FUNCTION_BLOCK ASR_CLIENT_0 (* Trigger 2 independent remote OPC-UA method calls via CLIENT_0, driven by an ASR adapter Socket (Set/Reset) *)
  (* Standard: 61499-2; Description: Copyright (c) 2026 HR Agrartechnik GmbH This program and the accompanying materials are made available under the terms of the Eclipse Public License 2.0 which is available at https://www.eclipse.org/legal/epl-2.0/ SPDX-License-Identifier: EPL-2.0 *)
  (* Version 1.0, 2026-09-03, Franz Höpfinger, HR Agrartechnik GmbH, initial API and implementation and/or initial documentation *)
  PACKAGE adapter::net;
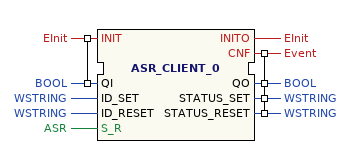
  EVENT_INPUT
    INIT : EInit WITH QI; (* Initialization *)
  END_EVENT
  EVENT_OUTPUT
    INITO : EInit; (* Initialization Confirm *)
    CNF WITH QO, STATUS_SET, STATUS_RESET; (* QO/STATUS updated *)
  END_EVENT
  VAR_INPUT
    QI : BOOL;
    ID_SET : WSTRING; (* Remote-Methodenadresse fuer den Set-Aufruf *)
    ID_RESET : WSTRING; (* Remote-Methodenadresse fuer den Reset-Aufruf *)
  END_VAR
  VAR_OUTPUT
    QO : BOOL; (* TRUE nur wenn SET_CLIENT und RESET_CLIENT aktuell beide QO=TRUE melden *)
    STATUS_SET : WSTRING; (* STATUS von SET_CLIENT *)
    STATUS_RESET : WSTRING; (* STATUS von RESET_CLIENT *)
  END_VAR
  SOCKETS
    S_R : adapter::types::unidirectional::ASR; (* Set/Reset *)
  END_SOCKETS
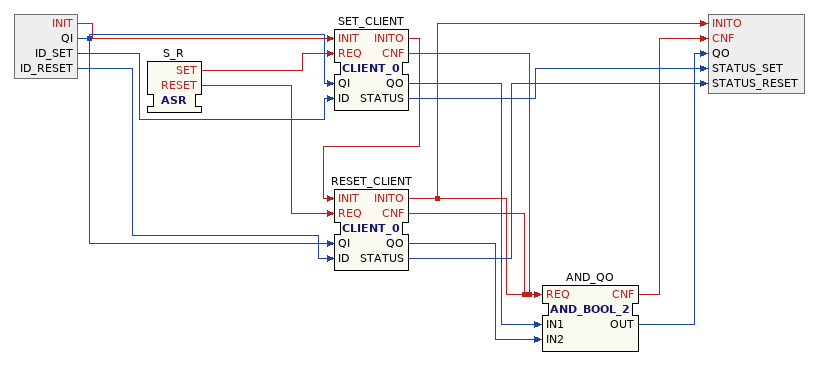
  FBS
    SET_CLIENT : iec61499::net::CLIENT_0;
    RESET_CLIENT : iec61499::net::CLIENT_0;
    AND_QO : iec61131::booleanOperators::AND_BOOL_2;
  END_FBS
  EVENT_CONNECTIONS
    INIT TO SET_CLIENT.INIT;
    SET_CLIENT.INITO TO RESET_CLIENT.INIT;
    RESET_CLIENT.INITO TO INITO;
    RESET_CLIENT.INITO TO AND_QO.REQ;
    S_R.SET TO SET_CLIENT.REQ;
    S_R.RESET TO RESET_CLIENT.REQ;
    SET_CLIENT.CNF TO AND_QO.REQ;
    RESET_CLIENT.CNF TO AND_QO.REQ;
    AND_QO.CNF TO CNF;
  END_CONNECTIONS
  DATA_CONNECTIONS
    QI TO SET_CLIENT.QI;
    QI TO RESET_CLIENT.QI;
    ID_SET TO SET_CLIENT.ID;
    ID_RESET TO RESET_CLIENT.ID;
    SET_CLIENT.QO TO AND_QO.IN1;
    RESET_CLIENT.QO TO AND_QO.IN2;
    AND_QO.OUT TO QO;
    SET_CLIENT.STATUS TO STATUS_SET;
    RESET_CLIENT.STATUS TO STATUS_RESET;
  END_CONNECTIONS
END_FUNCTION_BLOCK
